Staubli VAL3: find.pgx

public program find(string& x_sItem[], bool& x_bFound[])
begin
  //
  // find one item in the list
  //
end
